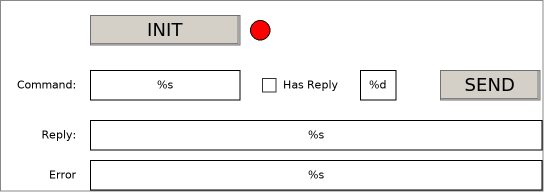
VISUALIZATION GUI_TEMPLATE_USB_COMM  // 544x192
VAR_IN_OUT
	m_Instance:	FB_ADS_COMM;
END_VAR
VAR
	cmd:			STRING;
	bHasReply:		BOOL;		(* If TRUE, there is a reply to the command *)
	nNumReplies:	DINT;	(* Number of replies, i.e. number of cfg.sReplySuffix strings expected in the reply *)
END_VAR
    Button (440,70 100x30), "SEND"
        OnMouseClick: execute {
            m_Instance.ctrl.nCommand:=2;
            m_Instance.ctrl.sCmd:=cmd;
            m_Instance.ctrl.bHasReply:=bHasReply;
            m_Instance.ctrl.nNumReplies:=nNumReplies;
            m_Instance.ctrl.bExecute:=TRUE;
        }
    Rectangle (90,120 452x30), "%s", text variable: m_Instance.stat.sReply
    Rectangle (90,70 150x30), "%s", tooltip "Command (without terminators)", text variable: cmd
        OnMouseClick: write the text variable via Default
    Button (90,15 150x30), "INIT", tooltip "Initialize communication"
        OnMouseClick: execute { m_Instance.ctrl.nCommand:=1; m_Instance.ctrl.bExecute:=TRUE; }
    Checkbox (260,70 97x30), "Has Reply", tooltip "Check this box if reply is expected", variable: bHasReply
    Rectangle (360,70 36x30), "%d", tooltip "Set the number of expected replies", text variable: nNumReplies, input disabled if: FALSE
        OnMouseClick: write the text variable via Default, min 0
    Label (10,70 69x30), "Command:"
    Label (10,120 69x30), "Reply:"
    Label (10,160 69x30), "Error"
    Rectangle (90,160 452x30), "%s", text variable: m_Instance.stat.sErrorText
    Ellipse (250,20 20x20), tooltip "GREEN=Initialized RED=Not-initialized", text variable: m_Instance.stat.bInitialised, colour toggle: m_Instance.stat.bInitialised
END_VISUALIZATION

(* stored: Version 1.1.0.1, ProductVersion 3.1.4024.3
   Visu GUI_TEMPLATE_USB_COMM: Id {256e685d-5e0a-4fb8-896b-b3e605c45e15} *)
